FUNCTION_BLOCK Database
VAR_INPUT
END_VAR
VAR_OUTPUT
END_VAR
VAR
END_VAR

END_FUNCTION_BLOCK

(* stored: Version 1.1.0.1, ProductVersion 3.1.4024.9
   POU Database: Id {605d332b-7be9-43a5-a170-f4dde6c122d7}, SpecialFunc None *)
